FUNCTION_BLOCK EC_START_ELEM (* Starts the instance of a FB, Connection (Event/Data), Resource or Device according to the state machine of IEC 61499 FBs *)
  (* Standard: 61499-1; Classification: Reconfiguration; Function: Starts FB, Connection, Resource or Device instances; Type: Execution Control Service; Description: Copyright (c) 2012 Profactor GmbH This program and the accompanying materials are made available under the terms of the Eclipse Public License 2.0 which is available at https://www.eclipse.org/legal/epl-2.0/ SPDX-License-Identifier: EPL-2.0 *)
  (* Version 1.0, 2012-05-31, Gerhard Ebenhofer, Profactor GmbH *)
  (* Compiler Cpp GNU GCC >3.0 *)
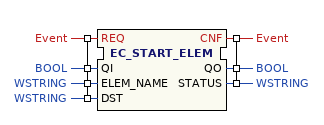
  EVENT_INPUT
    REQ WITH ELEM_NAME, DST, QI; (* Event to require starting an element *)
  END_EVENT
  EVENT_OUTPUT
    CNF WITH STATUS, QO; (* Event to confirm that the element has been started *)
  END_EVENT
  VAR_INPUT
    QI : BOOL; (* Event Input Qualifier *)
    ELEM_NAME : WSTRING; (* Element instance name *)
    DST : WSTRING; (* Destination where the element has to be started (Syntax: ResourceName) *)
  END_VAR
  VAR_OUTPUT
    QO : BOOL; (* Event Output Qualifier *)
    STATUS : WSTRING; (* Service Status: RDY, NO_SUCH_OBJECT, INVALID_STATE *)
  END_VAR
  SERVICE APPLICATION/RESOURCE (* Starts the instance of a FB, Connection (Event/Data), Resource or Device according to the state machine of IEC 61499 FBs *)
    SEQUENCE normal_establishment
      APPLICATION.INIT+() -> APPLICATION.INITO+();
    END_SEQUENCE
    SEQUENCE unsuccessful_establishment
      APPLICATION.INIT+() -> APPLICATION.INITO-();
    END_SEQUENCE
    SEQUENCE request_confirm
      APPLICATION.REQ+() -> APPLICATION.CNF+();
    END_SEQUENCE
    SEQUENCE request_inhibited
      APPLICATION.REQ-() -> APPLICATION.CNF-();
    END_SEQUENCE
    SEQUENCE request_error
      APPLICATION.REQ+() -> APPLICATION.CNF-();
    END_SEQUENCE
    SEQUENCE application_initiated_termination
      APPLICATION.INIT-() -> APPLICATION.INITO-();
    END_SEQUENCE
    SEQUENCE resource_initiated_termination
      -> APPLICATION.INITO-();
    END_SEQUENCE
  END_SERVICE
END_FUNCTION_BLOCK
